KUKA KRL data list: hp248.dat

&ACCESS RVP
&REL 17
&COMMENT Limpeza
&PARAM TEMPLATE = C:\KRC\roboter\template\vg_hp
&PARAM EDITMASK = HP*
DEFDAT HP248
;FOLD EXTERNAL DECLARATIONS;%{PE}%MKUKATPBASIS,%CEXT,%VCOMMON,%P
 ;FOLD BASISTECH EXT;%{PE}%MKUKATPBASIS,%CEXT,%VEXT,%P
   EXT  BAS (BAS_COMMAND  :IN,REAL  :IN )
   DECL INT SUCCESS
 ;ENDFOLD (BASISTECH EXT)
 ;FOLD GRIPPERTECH EXT
   EXT  H50 (INT:IN, INT:IN ,INT:IN ,GRP_TYP:IN)
 ;ENDFOLD (GRIPPERTECH EXT)
 ;FOLD SPOTTECH EXT
   EXT  USERSPOT (S_COMMAND  :IN, SPOT_TYPE:IN)
 ;ENDFOLD (SPOTTECH EXT)
 ;FOLD USER EXT;%{E}%MKUKATPUSER,%CEXT,%VEXT,%P
 ;Make here your modifications

  ;FOLD COLLISION
    EXT COLLSTOP(INT:IN,INT:IN)
  ;ENDFOLD  (Collision)
 ;ENDFOLD (USER EXT)
;ENDFOLD (EXTERNAL DECLERATIONS)
DECL FDAT FHOME={TOOL_NO 0,BASE_NO 0,IPO_FRAME #BASE}
ENDDAT
